// TIA Portal V20 export
FUNCTION_BLOCK "Simulation"   // FB195, LAD
// stored: MemoryReserve 100, Namespace Unit1.Em13, SetENOAutomatically false
   VAR_INPUT
      simulation { ExternalAccessible := 'False'; ExternalVisible := 'False'; ExternalWritable := 'False'} : Bool;
   END_VAR
   VAR
      instActuator { ExternalAccessible := 'False'; ExternalVisible := 'False'; ExternalWritable := 'False'} : Array[0..9] of "Simulation_Actuator";
      statDigitalSignal { ExternalAccessible := 'False'; ExternalVisible := 'False'; ExternalWritable := 'False'} : Array[0..9] of Bool;
   END_VAR
   VAR_TEMP   // added for the SCL form of the ladder/FBD networks
      _w1 : Bool;
   END_VAR
BEGIN

REGION Network 1: Digital Signal
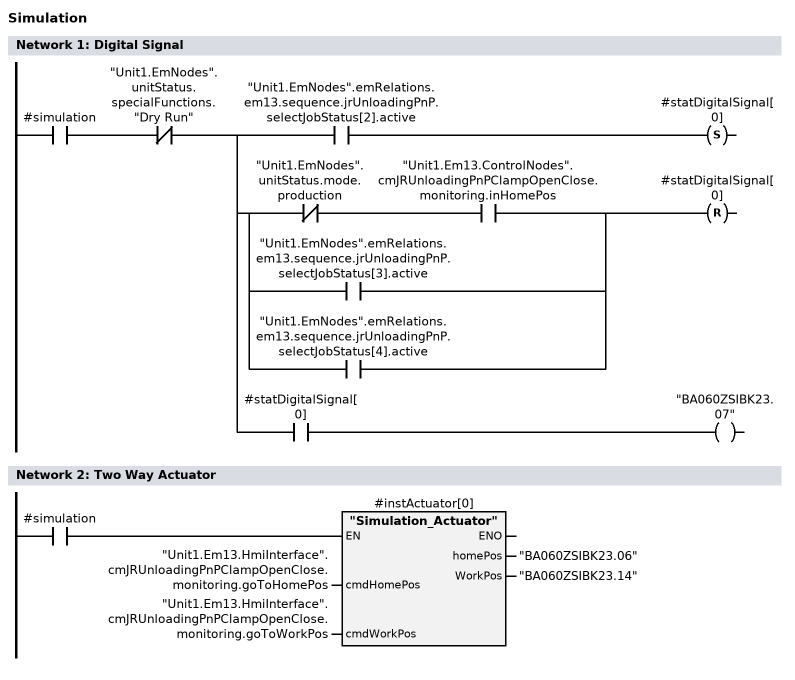
   RUNG wire#powerrail
      Contact( #simulation )
      I_Contact( "Unit1.EmNodes".unitStatus.specialFunctions."Dry Run" )
      wire#w1
      Contact( "Unit1.EmNodes".emRelations.em13.sequence.jrUnloadingPnP.selectJobStatus[2].active )
      S_Coil( #statDigitalSignal[0] )
   END_RUNG
   RUNG wire#w1
      I_Contact( "Unit1.EmNodes".unitStatus.mode.production )
      Contact( "Unit1.Em13.ControlNodes".cmJRUnloadingPnPClampOpenClose.monitoring.inHomePos )
      wire#w2
      R_Coil( #statDigitalSignal[0] )
   END_RUNG
   RUNG wire#w1
      Contact( "Unit1.EmNodes".emRelations.em13.sequence.jrUnloadingPnP.selectJobStatus[3].active )
   END_RUNG wire#w2
   RUNG wire#w1
      Contact( "Unit1.EmNodes".emRelations.em13.sequence.jrUnloadingPnP.selectJobStatus[4].active )
   END_RUNG wire#w2
   RUNG wire#w1
      Contact( #statDigitalSignal[0] )
      Coil( "BA060ZSIBK23.07" )
   END_RUNG
   // the same network as SCL:
   #_w1 := #simulation AND NOT "Unit1.EmNodes".unitStatus.specialFunctions."Dry Run";
   IF #_w1 AND "Unit1.EmNodes".emRelations.em13.sequence.jrUnloadingPnP.selectJobStatus[2].active THEN
       #statDigitalSignal[0] := TRUE;
   END_IF;
   IF #_w1 AND ((NOT "Unit1.EmNodes".unitStatus.mode.production AND "Unit1.Em13.ControlNodes".cmJRUnloadingPnPClampOpenClose.monitoring.inHomePos) OR "Unit1.EmNodes".emRelations.em13.sequence.jrUnloadingPnP.selectJobStatus[3].active OR "Unit1.EmNodes".emRelations.em13.sequence.jrUnloadingPnP.selectJobStatus[4].active) THEN
       #statDigitalSignal[0] := FALSE;
   END_IF;
   "BA060ZSIBK23.07" := #_w1 AND #statDigitalSignal[0];
END_REGION

REGION Network 2: Two Way Actuator
   RUNG wire#powerrail
      Contact( #simulation )
      #instActuator[0](cmdHomePos := "Unit1.Em13.HmiInterface".cmJRUnloadingPnPClampOpenClose.monitoring.goToHomePos, cmdWorkPos := "Unit1.Em13.HmiInterface".cmJRUnloadingPnPClampOpenClose.monitoring.goToWorkPos, homePos => "BA060ZSIBK23.06", WorkPos => "BA060ZSIBK23.14")
   END_RUNG
   // the same network as SCL:
   IF #simulation THEN
       #instActuator[0](cmdHomePos := "Unit1.Em13.HmiInterface".cmJRUnloadingPnPClampOpenClose.monitoring.goToHomePos,   // "Simulation_Actuator"
                        cmdWorkPos := "Unit1.Em13.HmiInterface".cmJRUnloadingPnPClampOpenClose.monitoring.goToWorkPos,
                        homePos => "BA060ZSIBK23.06",
                        WorkPos => "BA060ZSIBK23.14");
   END_IF;
END_REGION

REGION Network 3 (SCL): homing



   IF #simulation AND "JB_Temp".Test_Homing[13] THEN


       "Unit1.Em13.HmiInterface".cmJRUnloadingPnPClampOpenClose.commands.commandHomePos :=

       "Unit1.Em13.HmiInterface".cmJRUnloadingPnPAxisX.commands.homing :=
       "Unit1.Em13.HmiInterface".cmJRUnloadingPnPAxisZ.commands.homing :=
       "Unit1.Em13.HmiInterface".cmJRUnloadingPnPAxisC.commands.homing := true;


       "JB_Temp".Test_Homing[13] := false;
    //   
   END_IF;

   IF #simulation AND "JB_Temp".Test_Homing[20] THEN


       "Unit1.Em13.HmiInterface".cmJRUnloadingPnPAxisX.commands.homing :=
       "Unit1.Em13.HmiInterface".cmJRUnloadingPnPAxisZ.commands.homing :=
       "Unit1.Em13.HmiInterface".cmJRUnloadingPnPAxisC.commands.homing := FALSE;


       "JB_Temp".Test_Homing[20] := false;
   END_IF;


   "JB_Temp".Test_Homing[20] := "JB_Temp".Simulation_initializing;
   "JB_Temp".Simulation_initializing := false;
END_REGION
END_FUNCTION_BLOCK
